KUKA KRL program: tunegripper.src, tunegripper.dat

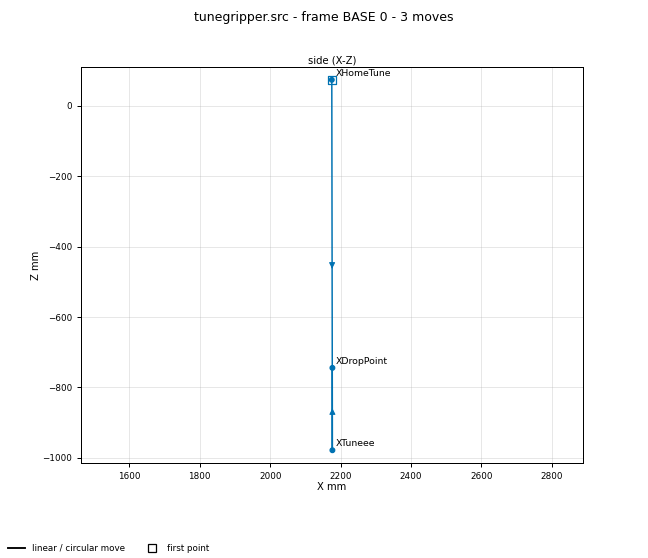
[picture p0: tool path of tunegripper.src in frame BASE 0, 3 of 3 moves have a stored position in this frame; points joined in program order, loops and branches not executed]
--- tunegripper.src ---
&ACCESS RVP
&REL 24
&PARAM EDITMASK = *
&PARAM TEMPLATE = C:\KRC\Roboter\Template\vorgabe
&PARAM DISKPATH = KRC:\R1\Program\Palletize
DEF TuneGripper( )
;FOLD INI;%{PE}
  ;FOLD BASISTECH INI
    GLOBAL INTERRUPT DECL 3 WHEN $STOPMESS==TRUE DO IR_STOPM ( )
    INTERRUPT ON 3
    BAS (#INITMOV,0 )
  ;ENDFOLD (BASISTECH INI)
;FOLD SPOTTECH INI
USERSPOT(#INIT)
;ENDFOLD (SPOTTECH INI)
;FOLD GRIPPERTECH INI
USER_GRP(0,DUMMY,DUMMY,GDEFAULT)
;ENDFOLD (GRIPPERTECH INI)
  ;FOLD USER INI
    ;Make your modifications here

  ;ENDFOLD (USER INI)
;ENDFOLD (INI)

;FOLD PTP HomeTune Vel=100 % PDAT2 Tool[1] Base[0];%{PE}%R 8.3.31,%MKUKATPBASIS,%CMOVE,%VPTP,%P 1:PTP, 2:HomeTune, 3:, 5:100, 7:PDAT2
$BWDSTART=FALSE
PDAT_ACT=PPDAT2
FDAT_ACT=FHomeTune
BAS(#PTP_PARAMS,100)
PTP XHomeTune
;ENDFOLD

loop
;FOLD SYN OUT 19 'RighPusGrpExt' State=FALSE at START Delay=0 ms;%{PE}%R 8.3.31,%MKUKATPBASIS,%COUT,%VSYNOUT,%P 2:19, 3:RighPusGrpExt, 5:FALSE, 7:0, 9:0, 12:0
TRIGGER WHEN DISTANCE=0 DELAY=0 DO $OUT[19]=FALSE
;ENDFOLD
;FOLD SYN OUT 26 'LeftPusGrpRec' State=FALSE at START Delay=0 ms;%{PE}%R 8.3.31,%MKUKATPBASIS,%COUT,%VSYNOUT,%P 2:26, 3:LeftPusGrpRec, 5:FALSE, 7:0, 9:0, 12:0
TRIGGER WHEN DISTANCE=0 DELAY=0 DO $OUT[26]=FALSE
;ENDFOLD
;FOLD SYN OUT 20 'RighPusGrpRec' State=TRUE at START Delay=0 ms;%{PE}%R 8.3.31,%MKUKATPBASIS,%COUT,%VSYNOUT,%P 2:20, 3:RighPusGrpRec, 5:TRUE, 7:0, 9:0, 12:0
TRIGGER WHEN DISTANCE=0 DELAY=0 DO $OUT[20]=TRUE
;ENDFOLD
;FOLD SYN OUT 25 'LeftPusGrpExt' State=TRUE at START Delay=0 ms;%{PE}%R 8.3.31,%MKUKATPBASIS,%COUT,%VSYNOUT,%P 2:25, 3:LeftPusGrpExt, 5:TRUE, 7:0, 9:0, 12:0
TRIGGER WHEN DISTANCE=0 DELAY=0 DO $OUT[25]=TRUE
;ENDFOLD
;Flg
$out[18] = false
$out[28] = false
$out[17] = true
$out[27] = true

;PLA
$out[24] = false
$out[22] = false
$out[23] = true
$out[21] = true

;FOLD WAIT Time=2 sec;%{PE}%R 8.3.31,%MKUKATPBASIS,%CWAIT,%VWAIT,%P 3:2
WAIT SEC 2
;ENDFOLD
;FOLD LIN Tuneee Vel=2 m/s CPDAT4 Tool[1] Base[0];%{PE}%R 8.3.31,%MKUKATPBASIS,%CMOVE,%VLIN,%P 1:LIN, 2:Tuneee, 3:, 5:2, 7:CPDAT4
$BWDSTART=FALSE
LDAT_ACT=LCPDAT4
FDAT_ACT=FTuneee
BAS(#CP_PARAMS,2)
LIN XTuneee
;ENDFOLD

wait sec 1.5

;PLA
$out[23] = false
$out[21] = false
$out[24] = true
$out[22] = true


;Flg
$out[17] = false
$out[27] = false
$out[18] = true
$out[28] = true


wait sec 2
   ;FOLD SYN OUT 20 'RighPusGrpRec' State=FALSE at START Delay=0 ms;%{PE}%R 8.3.31,%MKUKATPBASIS,%COUT,%VSYNOUT,%P 2:20, 3:RighPusGrpRec, 5:TRUE, 7:0, 9:0, 12:0
TRIGGER WHEN DISTANCE=0 DELAY=1000 DO $OUT[20]=FALSE
;ENDFOLD
;FOLD SYN OUT 25 'LeftPusGrpExt' State=FALSE at START Delay=0 ms;%{PE}%R 8.3.31,%MKUKATPBASIS,%COUT,%VSYNOUT,%P 2:25, 3:LeftPusGrpExt, 5:TRUE, 7:0, 9:0, 12:0
TRIGGER WHEN DISTANCE=0 DELAY=1000 DO $OUT[25]=FALSE
;ENDFOLD
   ;FOLD SYN OUT 19 'RighPusGrpExt' State=TRUE at START Delay=0 ms;%{PE}%R 8.3.31,%MKUKATPBASIS,%COUT,%VSYNOUT,%P 2:19, 3:RighPusGrpExt, 5:FALSE, 7:0, 9:0, 12:0
TRIGGER WHEN DISTANCE=0 DELAY=1000 DO $OUT[19]=TRUE
;ENDFOLD
;FOLD SYN OUT 26 'LeftPusGrpRec' State=TRUE at START Delay=0 ms;%{PE}%R 8.3.31,%MKUKATPBASIS,%COUT,%VSYNOUT,%P 2:26, 3:LeftPusGrpRec, 5:FALSE, 7:0, 9:0, 12:0
TRIGGER WHEN DISTANCE=0 DELAY=1000 DO $OUT[26]=TRUE
;ENDFOLD

;FOLD LIN DropPoint Vel=2 m/s CPDAT3 Tool[1] Base[0];%{PE}%R 8.3.31,%MKUKATPBASIS,%CMOVE,%VLIN,%P 1:LIN, 2:DropPoint, 3:, 5:2, 7:CPDAT3
$BWDSTART=FALSE
LDAT_ACT=LCPDAT3
FDAT_ACT=FDropPoint
BAS(#CP_PARAMS,2)
LIN XDropPoint
;ENDFOLD

ENDLOOP

end

--- tunegripper.dat ---
&ACCESS RVP
&REL 24
&PARAM EDITMASK = *
&PARAM TEMPLATE = C:\KRC\Roboter\Template\vorgabe
&PARAM DISKPATH = KRC:\R1\Program\Palletize
DEFDAT  tunegripper
;FOLD EXTERNAL DECLARATIONS;%{PE}%MKUKATPBASIS,%CEXT,%VCOMMON,%P
;FOLD GRIPPERTECH EXT
  EXT  H50 (INT:IN, INT:IN ,INT:IN ,GRP_TYP:IN)
;ENDFOLD (GRIPPERTECH EXT)
;FOLD SPOTTECH EXT
  EXT  USERSPOT (S_COMMAND  :IN, SPOT_TYPE:IN)
;ENDFOLD (SPOTTECH EXT)
;FOLD BASISTECH EXT;%{PE}%MKUKATPBASIS,%CEXT,%VEXT,%P
EXT  BAS (BAS_COMMAND  :IN,REAL  :IN )
DECL INT SUCCESS
;ENDFOLD (BASISTECH EXT)
;FOLD USER EXT;%{E}%MKUKATPUSER,%CEXT,%VEXT,%P
;Make your modifications here

;ENDFOLD (USER EXT)
;ENDFOLD (EXTERNAL DECLARATIONS)
DECL BASIS_SUGG_T LAST_BASIS={POINT1[] "Tuneee                  ",POINT2[] "Tuneee                  ",CP_PARAMS[] "CPDAT4                  ",PTP_PARAMS[] "PDAT3                   ",CONT[] "                        ",CP_VEL[] "2                       ",PTP_VEL[] "100                     ",SYNC_PARAMS[] "SYNCDAT                 ",SPL_NAME[] "S0                      ",A_PARAMS[] "ADAT0                   "}
DECL E6POS XTUNEPOSITION={X 2175.01318,Y -676.199829,Z -395.064758,A -0.880975723,B 0.212102517,C 178.762634,S 2,T 34,E1 0.0,E2 0.0,E3 0.0,E4 0.0,E5 0.0,E6 0.0}
DECL FDAT FTunePosition={TOOL_NO 1,BASE_NO 0,IPO_FRAME #BASE,POINT2[] " ",TQ_STATE FALSE}
DECL PDAT PPDAT1={VEL 100.000,ACC 100.000,APO_DIST 100.000,GEAR_JERK 50.0000}
DECL E6POS XHOMETUNE={X 2175.01318,Y -676.199829,Z 73.8199158,A -0.880975723,B 0.212102503,C 178.762634,S 2,T 34,E1 0.0,E2 0.0,E3 0.0,E4 0.0,E5 0.0,E6 0.0}
DECL FDAT FHomeTune={TOOL_NO 1,BASE_NO 0,IPO_FRAME #BASE,POINT2[] " ",TQ_STATE FALSE}
DECL PDAT PPDAT2={VEL 100.000,ACC 100.000,APO_DIST 100.000,GEAR_JERK 50.0000}
DECL E6POS XDROPPOINT={X 2176.73486,Y -676.199829,Z -744.270752,A -1.56035709,B 0.212195322,C 178.768677,S 2,T 34,E1 0.0,E2 0.0,E3 0.0,E4 0.0,E5 0.0,E6 0.0}
DECL FDAT FDropPoint={TOOL_NO 1,BASE_NO 0,IPO_FRAME #BASE,POINT2[] " ",TQ_STATE FALSE}
DECL LDAT LCPDAT1={VEL 2.00000,ACC 100.000,APO_DIST 100.000,APO_FAC 50.0000,AXIS_VEL 100.000,AXIS_ACC 100.000,ORI_TYP #VAR,CIRC_TYP #BASE,JERK_FAC 50.0000,GEAR_JERK 50.0000,EXAX_IGN 0}
DECL PDAT PPDAT3={VEL 100.000,ACC 100.000,APO_DIST 100.000,GEAR_JERK 50.0000}
DECL LDAT LCPDAT2={VEL 2.00000,ACC 100.000,APO_DIST 100.000,APO_FAC 50.0000,AXIS_VEL 100.000,AXIS_ACC 100.000,ORI_TYP #VAR,CIRC_TYP #BASE,JERK_FAC 50.0000,GEAR_JERK 50.0000,EXAX_IGN 0}
DECL LDAT LCPDAT3={VEL 2.00000,ACC 100.000,APO_DIST 100.000,APO_FAC 50.0000,AXIS_VEL 100.000,AXIS_ACC 100.000,ORI_TYP #VAR,CIRC_TYP #BASE,JERK_FAC 50.0000,GEAR_JERK 50.0000,EXAX_IGN 0}
DECL E6POS XTUNEEE={X 2176.73486,Y -676.199829,Z -978.265381,A -1.56035721,B 0.212195367,C 178.768677,S 2,T 34,E1 0.0,E2 0.0,E3 0.0,E4 0.0,E5 0.0,E6 0.0}
DECL FDAT FTuneee={TOOL_NO 1,BASE_NO 0,IPO_FRAME #BASE,POINT2[] " ",TQ_STATE FALSE}
DECL LDAT LCPDAT4={VEL 2.00000,ACC 100.000,APO_DIST 100.000,APO_FAC 50.0000,AXIS_VEL 100.000,AXIS_ACC 100.000,ORI_TYP #VAR,CIRC_TYP #BASE,JERK_FAC 50.0000,GEAR_JERK 50.0000,EXAX_IGN 0}
ENDDAT
